// Mitsubishi GX Works2 project: festotest   PLC: Q03UDE

PROGRAM MAIN
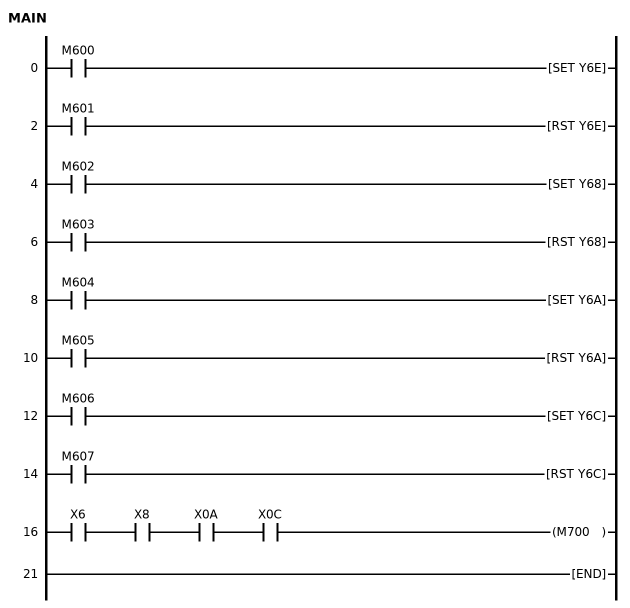
0     LD      M600
      SET     Y6E
2     LD      M601
      RST     Y6E
4     LD      M602
      SET     Y68
6     LD      M603
      RST     Y68
8     LD      M604
      SET     Y6A
10    LD      M605
      RST     Y6A
12    LD      M606
      SET     Y6C
14    LD      M607
      RST     Y6C
16    LD      X6
      AND     X8
      AND     X0A
      AND     X0C
      OUT     M700
21    END
END_PROGRAM
